// TIA Portal V17 export
// export: Created 2026-04-13T11:12:44.6157173Z, ExportSetting WithDefaults, DisplayName Totally Integrated Automation Portal, DisplayVersion V17 Update 4, DisplayName TIA Portal Openness, DisplayVersion V17 Update 4, DisplayName TIA Portal Version Control Interface, DisplayVersion V17, DisplayName SINAMICS Startdrive Advanced, DisplayVersion V17, DisplayName SINAMICS Startdrive G130, G150, S120, S150, SINAMICS MV, S210, DisplayVersion V17, DisplayName SINAMICS Startdrive G110M, G120, G120C, G120D, G120P, G115D, DisplayVersion V17, DisplayName STEP 7 Professional, DisplayVersion V17 Update 4, DisplayName STEP 7 Safety, DisplayVersion V17, DisplayName WinCC Professional, DisplayVersion V17 Update 4
DATA_BLOCK "C4-室外CIP清洗_DB"   // DB31
VERSION : 0.1
// stored: AutoNumber true, DBAccessibleFromOPCUA true, DBAccessibleFromWebserver true, InstanceOfName C4-室外CIP清洗, InstanceOfType FB
"C4-室外CIP清洗"
   // VAR
   //    室外CIP清洗 { S7_SetPoint := 'True'} : "OUTCIP清洗";
   //    FT1 { S7_SetPoint := 'True'} : F_TRIG;
   //    FT2 { S7_SetPoint := 'True'} : F_TRIG;
   //    FT3 { S7_SetPoint := 'True'} : F_TRIG;
   //    TON1 { S7_SetPoint := 'True'} : TON_TIME;
   //    PT1 { S7_SetPoint := 'True'} : Time;
   //    T1S : TON_TIME;
   //    YC1 { S7_SetPoint := 'True'} : DInt;
   //    YC2 : DInt;
   //    YC3 : DInt;
   //    TP1 : Bool;
   //    TP2 : Bool;
   //    TP3 : Bool;
   //    T_10HZ : TON_TIME;
   //    GET_Instance { S7_SetPoint := 'True'} : GET;
   //    PUT_Instance { S7_SetPoint := 'True'} : PUT;
   // END_VAR
BEGIN
END_DATA_BLOCK
